FUNCTION F_PistonDisplacementToBoomAngle : LREAL
VAR_INPUT
	xCyl : LREAL;
END_VAR
VAR
	AB : LREAL;
	AC : LREAL;
	BC : LREAL;
	alpha1 : LREAL;
	alpha2 : LREAL;
	theta1 : LREAL;
END_VAR

AB := SQRT(ABS(Parameters.stCraneKinematics.ABx)*ABS(Parameters.stCraneKinematics.ABx) + ABS(Parameters.stCraneKinematics.ABy)*ABS(Parameters.stCraneKinematics.ABy));
AC := SQRT(ABS(Parameters.stCraneKinematics.ACx)*ABS(Parameters.stCraneKinematics.ACx) + ABS(Parameters.stCraneKinematics.ACy)*ABS(Parameters.stCraneKinematics.ACy));

BC := 0.77222 + xCyl;

alpha1 := ATAN(ABS(Parameters.stCraneKinematics.ACy)/ ABS(Parameters.stCraneKinematics.ACx));
alpha2 := ATAN(ABS(Parameters.stCraneKinematics.ABy)/ ABS(Parameters.stCraneKinematics.ABx));

theta1 := ACOS( (ABS(AB)*ABS(AB) + ABS(AC)*ABS(AC) - (ABS(BC))*(ABS(AB)*ABS(AB) + ABS(AC)*ABS(AC) - (ABS(BC))) / (2 * ABS(AB) * ABS(AC)) ) - alpha2 + alpha1);

F_PistonDisplacementToBoomAngle := theta1;

END_FUNCTION

(* stored: Version 1.1.0.1, ProductVersion 3.1.4024.10
   POU F_PistonDisplacementToBoomAngle: Id {a235119c-45d2-4f49-b730-4da55738c20e}, SpecialFunc None *)
